{attribute 'GeneratedUsingTerminal: EPP6090-0000-0017'}
{attribute addProperty BoxType "EPP6090-0000-0017"}
{attribute addProperty Id "StatusAT %I*Status_E3E7FD126"}
{attribute addProperty CRC "3773007075"}
{attribute addProperty Size "6"}
TYPE DIS_Inputs_E0E384E3 :
STRUCT
	{attribute addProperty Name "Status"}
	Status AT %I* : Status_E3E7FD12;
END_STRUCT
END_TYPE

(* stored: Version 1.2.0.0, ProductVersion 3.1.4024.9
   DUT DIS_Inputs_E0E384E3: Id {d82d4b6f-edfe-4b60-9099-9b64a640d632} *)
